TYPE TcoUrRobotics_T2O_IO_IO :
STRUCT
    bArray AT %I* : ARRAY[0..67] OF BYTE;
END_STRUCT
END_TYPE

(* stored: Version 1.1.0.1, ProductVersion 3.1.4024.12
   DUT TcoUrRobotics_T2O_IO_IO: Id {df0d8ed2-b893-0bac-33d4-3efb3ce2f689} *)
